// Mitsubishi GX Works2 project: Deco_test   PLC: FX1S

PROGRAM MAIN
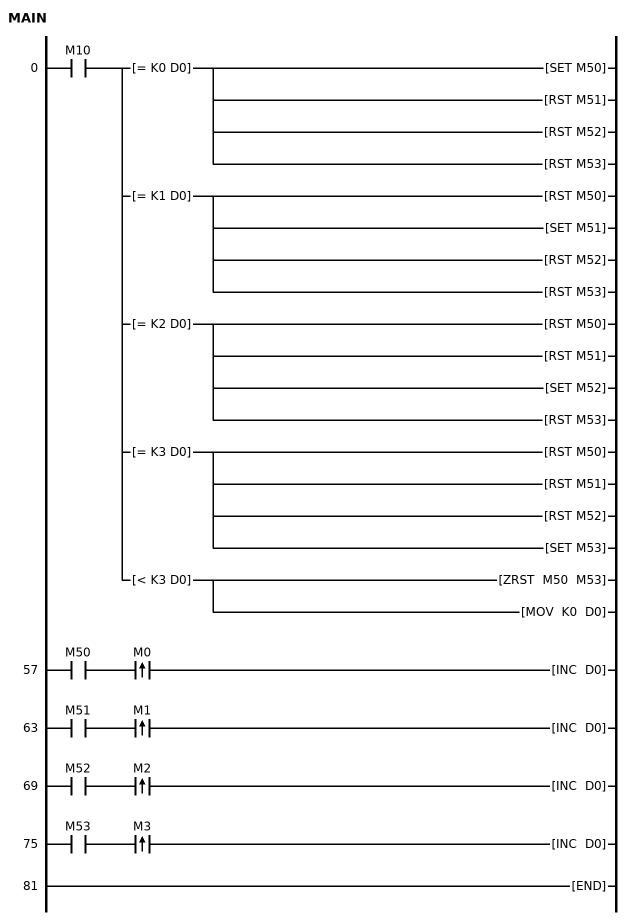
0     LD      M10
      MPS
      AND=    K0 D0
      SET     M50
      RST     M51
      RST     M52
      RST     M53
      MRD
      AND=    K1 D0
      RST     M50
      SET     M51
      RST     M52
      RST     M53
      MRD
      AND=    K2 D0
      RST     M50
      RST     M51
      SET     M52
      RST     M53
      MRD
      AND=    K3 D0
      RST     M50
      RST     M51
      RST     M52
      SET     M53
      MPP
      AND<    K3 D0
      ZRST    M50 M53
      MOV     K0 D0
57    LD      M50
      ANDP    M0
      INC     D0
63    LD      M51
      ANDP    M1
      INC     D0
69    LD      M52
      ANDP    M2
      INC     D0
75    LD      M53
      ANDP    M3
      INC     D0
81    END
END_PROGRAM
